PROGRAM Brouillon
VAR
END_VAR

END_PROGRAM

(* stored: Version 1.1.0.1
   POU Brouillon: Id {7b64cf9e-5d10-4cbb-81fd-348e1a12c5f2}, SpecialFunc None *)
